Staubli VAL3: centerCircle.pgx

public program centerCircle(point x_pFirst, point x_pMiddle, point x_pLast, trsf& x_tfCenter[], num& x_nRadius[])
  local frame l_frame
  local trsf tr[3]
  local num cx
  local num cy
begin
  x_tfCenter=x_pFirst.trsf
  l_frame=world
  setFrame(x_pFirst,x_pMiddle,x_pLast,l_frame)
  tr[0]=!l_frame.trsf*x_pFirst.trsf
  tr[1]=!l_frame.trsf*x_pLast.trsf
  tr[2]=!l_frame.trsf*x_pMiddle.trsf
  cy=0.5*(((tr[1].x-tr[2].x)*(tr[1].x/tr[1].y))+tr[1].y)
  cx=tr[2].x/2
  x_nRadius=sqrt((cx*cx)+(cy*cy))
  x_tfCenter=l_frame.trsf*{cx,cy,0,0,0,0}
  //tr[0]=!x_pCenter.trsf*x_pFirst.trsf
  //x_pCenter.trsf=x_pCenter.trsf*{0,0,0,0,0,atan(tr[0].y/tr[0].x)+180}
end
